# EPICS substitutions: bsaDriverApp/Db/bld.substitutions
file serviceChannelCtrl.db {
    pattern {   DEVICE,                  DESC,    SERVICE}
            {   "$(DEV)", "$(DESC\=\$\(SECN\))"  "BLD" }
}
